// TIA Portal V17 export
// export: Created 2025-03-05T08:02:20.1491544Z, ExportSetting WithDefaults, DisplayName Totally Integrated Automation Portal, DisplayVersion V17 Update 8, DisplayName TIA Portal Openness, DisplayVersion V17 Update 8, DisplayName TIA Portal Version Control Interface, DisplayVersion V17, DisplayName SINAMICS Startdrive Advanced, DisplayVersion V17 SP2, DisplayName SINAMICS Startdrive G110M, G120, G120C, G120D, G120P, G115D, DisplayVersion V17 SP2, DisplayName SINAMICS Startdrive G130, G150, S120, S150, SINAMICS MV, S210, DisplayVersion V17 SP2, DisplayName STEP 7 Professional, DisplayVersion V17 Update 8, DisplayName SINUMERIK ONE STEP 7 Toolbox, DisplayVersion V17 Update 12, DisplayName SINUMERIK 840D sl STEP 7 Toolbox, DisplayVersion V17 Update 12, DisplayName STEP 7 Safety, DisplayVersion V17 Update 6, DisplayName WinCC Advanced, DisplayVersion V17 Update 8
TYPE "GLOBAL_DATA_CLADDING"
// stored: IsFailsafeCompliant false
   STRUCT
      ALL_UNITS_RETURNED : Bool;   // ALL UNITS RETURNED
      ALL_UNITS_OUT_COLL_TRANSF : Bool;   // ALL UNITS OUT COLLISION TRANSFER
      ALL_STATIONS_UNIT_01_RETURNED : Bool;   // ALL UNITS RETURNED / ALL STATIONS UNIT 01 RETURNED
      ALL_STATIONS_UNIT_01_OUT_COLL_TRANSF : Bool;   // ALL UNIT OUT COLLISION TRANSFER / ALL STATIONS UNIT 01 OUT COLLISION TRANSFER
      ALL_STATIONS_UNIT_02_RETURNED : Bool;   // ALL UNITS RETURNED / ALL STATIONS UNIT 02 RETURNED
      ALL_STATIONS_UNIT_02_OUT_COLL_TRANSF : Bool;   // ALL UNIT OUT COLLISION TRANSFER / ALL STATIONS UNIT 02 OUT COLLISION TRANSFER
      ALL_CLAMPED_UNIT_01_ANALOG : Bool;   // ALL CLAMPED / ALL CLAMPED UNIT 01
      ALL_UNCLAMPED_UNIT_01_ANALOG : Bool;   // ALL UNCLAMPED / ALL UNCLAMPED UNIT 01
      ALL_CLAMPED_UNIT_02_ANALOG : Bool;   // ALL CLAMPED / ALL CLAMPED UNIT 02
      ALL_UNCLAMPED_UNIT_02_ANALOG : Bool;   // ALL UNCLAMPED / ALL UNCLAMPED UNIT 02
      CLAMPED_UNCLAMPED_UNIT_01_ANALOG : Bool;   // CLAMPED OR UNCLAMPED / CLAMPED OR UNCLAMPED UNIT 01
      CLAMPED_PARTIAL_CLAMPED_UNIT_01_ANALOG : Bool;   // CLAMPED OR UNCLAMPED / CLAMPED OR PARTIAL CLAMPED UNIT 01
      CLAMPED_UNCLAMPED_UNIT_02_ANALOG : Bool;   // CLAMPED OR UNCLAMPED / CLAMPED OR UNCLAMPED UNIT 02
      CLAMPED_PARTIAL_CLAMPED_UNIT_02_ANALOG : Bool;   // CLAMPED OR UNCLAMPED / CLAMPED OR PARTIAL CLAMPED UNIT 02
      ALL_CLAMPED_UNIT_01 : Bool;   // ALL CLAMPED / ALL CLAMPED UNIT 01
      ALL_UNCLAMPED_UNIT_01 : Bool;   // ALL UNCLAMPED / ALL UNCLAMPED UNIT 01
      ALL_CLAMPED_UNIT_02 : Bool;   // ALL CLAMPED / ALL CLAMPED UNIT 02
      ALL_UNCLAMPED_UNIT_02 : Bool;   // ALL UNCLAMPED / ALL UNCLAMPED UNIT 02
      CLAMPED_UNCLAMPED_UNIT_01 : Bool;   // CLAMPED OR UNCLAMPED / CLAMPED OR UNCLAMPED UNIT 01
      CLAMPED_PARTIAL_CLAMPED_UNIT_01 : Bool;   // CLAMPED OR UNCLAMPED / CLAMPED OR PARTIAL CLAMPED UNIT 01
      CLAMPED_UNCLAMPED_UNIT_02 : Bool;   // CLAMPED OR UNCLAMPED / CLAMPED OR UNCLAMPED UNIT 02
      CLAMPED_PARTIAL_CLAMPED_UNIT_02 : Bool;   // CLAMPED OR UNCLAMPED / CLAMPED OR PARTIAL CLAMPED UNIT 02
      CLAMPED_UNCLAMPED_UNIT_03 : Bool;   // CLAMPED OR UNCLAMPED / CLAMPED OR UNCLAMPED UNIT 03
      CLAMPED_PARTIAL_CLAMPED_UNIT_03 : Bool;   // CLAMPED OR UNCLAMPED / CLAMPED OR PARTIAL CLAMPED UNIT 03
      FIX_IN_UNIT_01_STA_1_UNCLAMPED_ANALOG : Bool;   // FIXTURE IN UNIT 01 LOAD UNLOAD STATION UNCLAMPED ANALOG
      FIX_IN_UNIT_01_STA_1_CLAMPED_ANALOG : Bool;   // FIXTURE IN UNIT 01 LOAD UNLOAD STATION CLAMPED ANALOG
      FIX_IN_UNIT_02_STA_1_UNCLAMPED_ANALOG : Bool;   // FIXTURE IN UNIT 02 LOAD UNLOAD STATION UNCLAMPED ANALOG
      FIX_IN_UNIT_02_STA_1_CLAMPED_ANALOG : Bool;   // FIXTURE IN UNIT 02 LOAD UNLOAD STATION CLAMPED ANALOG
      FIX_IN_UNIT_01_STA_2_UNCLAMPED_ANALOG : Bool;   // FIXTURE IN UNIT 01 SPARE STATION UNCLAMPED ANALOG
      FIX_IN_UNIT_01_STA_2_CLAMPED_ANALOG : Bool;   // FIXTURE IN UNIT 01 SPARE STATION CLAMPED ANALOG
      FIX_IN_UNIT_02_STA_2_UNCLAMPED_ANALOG : Bool;   // FIXTURE IN UNIT 02 SPARE STATION UNCLAMPED ANALOG
      FIX_IN_UNIT_02_STA_2_CLAMPED_ANALOG : Bool;   // FIXTURE UNIT 02 IN SPARE STATION CLAMPED ANALOG
      FIX_IN_UNIT_01_STA_3_UNCLAMPED_ANALOG : Bool;   // FIXTURE IN UNIT 01 CLADDING STATION UNCLAMPED ANALOG
      FIX_IN_UNIT_01_STA_3_CLAMPED_ANALOG : Bool;   // FIXTURE IN UNIT 01 CLADDING STATION CLAMPED ANALOG
      FIX_IN_UNIT_02_STA_3_UNCLAMPED_ANALOG : Bool;   // FIXTURE IN UNIT 02 CLADDING STATION UNCLAMPED ANALOG
      FIX_IN_UNIT_02_STA_3_CLAMPED_ANALOG : Bool;   // FIXTURE IN UNIT 02 CLADDING STATION CLAMPED ANALOG
      FIX_IN_UNIT_01_STA_4_UNCLAMPED_ANALOG : Bool;   // FIXTURE IN UNIT 01 MEASURING/CLEANING STATION UNCLAMPED ANALOG
      FIX_IN_UNIT_01_STA_4_CLAMPED_ANALOG : Bool;   // FIXTURE IN UNIT 01 MEASURING/CLEANING STATION CLAMPED ANALOG
      FIX_IN_UNIT_02_STA_4_UNCLAMPED_ANALOG : Bool;   // FIXTURE IN UNIT 02 MEASURING/CLEANING STATION UNCLAMPED ANALOG
      FIX_IN_UNIT_02_STA_4_CLAMPED_ANALOG : Bool;   // FIXTURE UNIT 02 IN MEASURING/CLEANING STATION CLAMPED ANALOG
      FIX_IN_UNIT_01_STA_1_UNCLAMPED : Bool;   // FIXTURE IN UNIT 01 LOAD UNLOAD STATION UNCLAMPED
      FIX_IN_UNIT_01_STA_1_CLAMPED : Bool;   // FIXTURE IN UNIT 01 LOAD UNLOAD STATION CLAMPED
      FIX_IN_UNIT_02_STA_1_UNCLAMPED : Bool;   // FIXTURE IN UNIT 02 LOAD UNLOAD STATION UNCLAMPED
      FIX_IN_UNIT_02_STA_1_CLAMPED : Bool;   // FIXTURE IN UNIT 02 LOAD UNLOAD STATION CLAMPED
      FIX_IN_UNIT_01_STA_2_UNCLAMPED : Bool;   // FIXTURE IN UNIT 01 SPARE STATION UNCLAMPED
      FIX_IN_UNIT_01_STA_2_CLAMPED : Bool;   // FIXTURE IN UNIT 01 SPARE STATION CLAMPED
      FIX_IN_UNIT_02_STA_2_UNCLAMPED : Bool;   // FIXTURE IN UNIT 02 SPARE STATION UNCLAMPED
      FIX_IN_UNIT_02_STA_2_CLAMPED : Bool;   // FIXTURE UNIT 02 IN SPARE STATION CLAMPED
      FIX_IN_UNIT_01_STA_3_UNCLAMPED : Bool;   // FIXTURE IN UNIT 01 CLADDING STATION UNCLAMPED
      FIX_IN_UNIT_01_STA_3_CLAMPED : Bool;   // FIXTURE IN UNIT 01 CLADDING STATION CLAMPED
      FIX_IN_UNIT_02_STA_3_UNCLAMPED : Bool;   // FIXTURE IN UNIT 02 CLADDING STATION UNCLAMPED
      FIX_IN_UNIT_02_STA_3_CLAMPED : Bool;   // FIXTURE IN UNIT 02 CLADDING STATION CLAMPED
      FIX_IN_UNIT_01_STA_4_UNCLAMPED : Bool;   // FIXTURE IN UNIT 01 MEASURING/CLEANING STATION UNCLAMPED
      FIX_IN_UNIT_01_STA_4_CLAMPED : Bool;   // FIXTURE IN UNIT 01 MEASURING/CLEANING STATION CLAMPED
      FIX_IN_UNIT_02_STA_4_UNCLAMPED : Bool;   // FIXTURE IN UNIT 02 MEASURING/CLEANING STATION UNCLAMPED
      FIX_IN_UNIT_02_STA_4_CLAMPED : Bool;   // FIXTURE UNIT 02 IN MEASURING/CLEANING STATION CLAMPED
      FIX_IN_UNIT_03_STA_MEAS_UNCLAMPED : Bool;   // FIXTURE IN UNIT 03 MEASURING STATION UNCLAMPED ANALOG
      FIX_IN_UNIT_03_STA_MEAS_CLAMPED : Bool;   // FIXTURE UNIT 03 IN MEASURING STATION CLAMPED ANALOG
      FIX_IN_UNIT_01_STA_0_ANY_CALIBRATION_MISS : Bool;   // FIXTURE IN UNIT 01 STATION 0 ANY CALIBRATION MISSING
      FIX_IN_UNIT_02_STA_0_ANY_CALIBRATION_MISS : Bool;   // FIXTURE IN UNIT 02 STATION 0 ANY CALIBRATION MISSING
      UNIT_01_ANY_FIX_CALIBRATION_MISS : Bool;   // UNIT 01 ANY FIXTURE CALIBRATION MISSING
      UNIT_02_ANY_FIX_CALIBRATION_MISS : Bool;   // UNIT 02 ANY FIXTURE CALIBRATION MISSING
      MACHINE_ANY_FIX_CALIBRATION_MISS : Bool;   // MACHINE ANY FIXTURE CALIBRATION MISSING
      ALL_FULL_DEPTH : Bool;   // ALL FULL DEPTH
      ALL_FULL_DEPTH_PULSE : Bool;   // ALL FULL DEPTH PULSE
      ALL_FULL_DEPTH_UNIT_01 : Bool;   // ALL FULL DEPTH / ALL FULL DEPTH UNIT 01
      ALL_FULL_DEPTH_PULSE_UNIT_01 : Bool;   // ALL FULL DEPTH PULSE / ALL FULL DEPTH PULSE UNIT 01
      ALL_FULL_DEPTH_UNIT_02 : Bool;   // ALL FULL DEPTH / ALL FULL DEPTH UNIT 02
      ALL_FULL_DEPTH_PULSE_UNIT_02 : Bool;   // ALL FULL DEPTH PULSE / ALL FULL DEPTH PULSE UNIT 02
      ALL_FULL_DEPTH_UNIT_03 : Bool;   // ALL FULL DEPTH / ALL FULL DEPTH UNIT 03
      ALL_FULL_DEPTH_PULSE_UNIT_03 : Bool;   // ALL FULL DEPTH PULSE / ALL FULL DEPTH PULSE UNIT 03
      RESET_FULL_DEPTH_UNIT_01_FIXT_1 : Bool;   // RESET FULL DEPTH / RESET FULL DEPTH UNIT 01 FIXTURE 1
      RESET_FULL_DEPTH_PULSE_UNIT_01_FIXT_1 : Bool;   // RESET FULL DEPTH PULSE / RESET FULL DEPTH PULSE UNIT 01 FIXTURE 1
      RESET_FULL_DEPTH_UNIT_01_FIXT_2 : Bool;   // RESET FULL DEPTH UNIT 01 FIXTURE 2
      RESET_FULL_DEPTH_PULSE_UNIT_01_FIXT_2 : Bool;   // RESET FULL DEPTH PULSE UNIT 01 FIXTURE 2
      RESET_FULL_DEPTH_UNIT_01_FIXT_3 : Bool;   // RESET FULL DEPTH / RESET FULL DEPTH UNIT 01 FIXTURE 3
      RESET_FULL_DEPTH_PULSE_UNIT_01_FIXT_3 : Bool;   // RESET FULL DEPTH PULSE / RESET FULL DEPTH PULSE UNIT 01 FIXTURE 3
      RESET_FULL_DEPTH_UNIT_01_FIXT_4 : Bool;   // RESET FULL DEPTH UNIT 01 FIXTURE 4
      RESET_FULL_DEPTH_PULSE_UNIT_01_FIXT_4 : Bool;   // RESET FULL DEPTH PULSE UNIT 01 FIXTURE 4
      RESET_FULL_DEPTH_UNIT_02_FIXT_1 : Bool;   // RESET FULL DEPTH / RESET FULL DEPTH UNIT 02 FIXTURE 1
      RESET_FULL_DEPTH_PULSE_UNIT_02_FIXT_1 : Bool;   // RESET FULL DEPTH PULSE / RESET FULL DEPTH PULSE UNIT 02 FIXTURE 1
      RESET_FULL_DEPTH_UNIT_02_FIXT_2 : Bool;   // RESET FULL DEPTH / RESET FULL DEPTH UNIT 02 FIXTURE 2
      RESET_FULL_DEPTH_PULSE_UNIT_02_FIXT_2 : Bool;   // RESET FULL DEPTH PULSE / RESET FULL DEPTH PULSE UNIT 02 FIXTURE 2
      RESET_FULL_DEPTH_UNIT_02_FIXT_3 : Bool;   // RESET FULL DEPTH / RESET FULL DEPTH UNIT 02 FIXTURE 3
      RESET_FULL_DEPTH_PULSE_UNIT_02_FIXT_3 : Bool;   // RESET FULL DEPTH PULSE / RESET FULL DEPTH PULSE UNIT 02 FIXTURE 3
      RESET_FULL_DEPTH_UNIT_02_FIXT_4 : Bool;   // RESET FULL DEPTH / RESET FULL DEPTH UNIT 02 FIXTURE 4
      RESET_FULL_DEPTH_PULSE_UNIT_02_FIXT_4 : Bool;   // RESET FULL DEPTH PULSE / RESET FULL DEPTH PULSE UNIT 02 FIXTURE 4
      RESET_FULL_DEPTH_UNIT_03_FIXT_1 : Bool;   // RESET FULL DEPTH / RESET FULL DEPTH UNIT 01 FIXTURE 1
      RESET_FULL_DEPTH_PULSE_UNIT_03_FIXT_1 : Bool;   // RESET FULL DEPTH PULSE / RESET FULL DEPTH PULSE UNIT 01 FIXTURE 1
      NO_MACHINE_CYCLE_RUN_P : Bool;   // NO CYCLE MACHINE RUN PROGRAM / NO MACHINE CYCLE RUNNING PULSE
      ANY_MACHINE_CYCLE_RUN_P : Bool;   // ANY MACHINE CYCLE RUN PROGRAM / ANY MACHINE CYCLE RUNNING PULSE
      NO_MACHINE_CYCLE_RUN_UNIT_01_P : Bool;   // NO CYCLE MACHINE RUN PROGRAM / NO MACHINE CYCLE RUNNING UNIT 01 PULSE
      ANY_UNIT_01_CYCLE_RUN_P : Bool;   // ANY MACHINE CYCLE RUN PROGRAM / ANY UNIT 01 CYCLE RUNNING PULSE
      NO_MACHINE_CYCLE_RUN_UNIT_02_P : Bool;   // NO CYCLE MACHINE RUN PROGRAM / NO MACHINE CYCLE RUNNING UNIT 02 PULSE
      ANY_UNIT_02_CYCLE_RUN_P : Bool;   // ANY MACHINE CYCLE RUN PROGRAM / ANY UNIT 02 CYCLE RUNNING PULSE
      NO_MACHINE_CYCLE_RUN_UNIT_03_P : Bool;   // NO CYCLE MACHINE RUN PROGRAM / NO MACHINE CYCLE RUNNING UNIT 03 PULSE
      ANY_UNIT_03_CYCLE_RUN_P : Bool;   // ANY MACHINE CYCLE RUN PROGRAM / ANY UNIT 03 CYCLE RUNNING PULSE
      NO_MACHINE_CYCLE_RUN_HOPPER_UNIT_01_P : Bool;   // NO CYCLE MACHINE RUN PROGRAM / NO MACHINE CYCLE RUNNING HOPPER UNIT 01 PULSE
      ANY_HOPPER_UNIT_01_CYCLE_RUN_P : Bool;   // ANY MACHINE CYCLE RUN PROGRAM / ANY HOPPER UNIT 01 CYCLE RUNNING PULSE
      NO_MACHINE_CYCLE_RUN_HOPPER_UNIT_02_P : Bool;   // NO CYCLE MACHINE RUN PROGRAM / NO MACHINE CYCLE RUNNING HOPPER UNIT 02 PULSE
      ANY_HOPPER_UNIT_02_CYCLE_RUN_P : Bool;   // ANY MACHINE CYCLE RUN PROGRAM / ANY HOPPER UNIT 02 CYCLE RUNNING PULSE
      FIX_IN_U_01_STA_1_ANY_FIX_SEQ_RUN : Bool;   // (GLOBAL BITS) COOLANT ON UNIT 01R / FIXTURE IN UNIT 01 STATION 1 RUNING ANY SEQUENCE
      FIX_IN_U_01_STA_2_ANY_FIX_SEQ_RUN : Bool;   // (GLOBAL BITS) COOLANT UNIT 01R WAIT FOR FILL TOOL / FIXTURE IN UNIT 01 STATION 2 RUNING ANY SEQUENCE
      FIX_IN_U_01_STA_3_ANY_FIX_SEQ_RUN : Bool;   // (GLOBAL BITS) COOLANT ON UNIT 01L / FIXTURE IN UNIT 01 STATION 3 RUNING ANY SEQUENCE
      FIX_IN_U_01_STA_4_ANY_FIX_SEQ_RUN : Bool;   // (GLOBAL BITS) COOLANT UNIT 01L WAIT FOR FILL TOOL / FIXTURE IN UNIT 01 STATION 4 RUNING ANY SEQUENCE
      FIX_IN_U_02_STA_1_ANY_FIX_SEQ_RUN : Bool;   // (GLOBAL BITS) COOLANT SP11 ON / FIXTURE IN UNIT 02 STATION 1 RUNING ANY SEQUENCE
      FIX_IN_U_02_STA_2_ANY_FIX_SEQ_RUN : Bool;   // (GLOBAL BITS) COOLANT SP12 ON / FIXTURE IN UNIT 02 STATION 2 RUNING ANY SEQUENCE
      FIX_IN_U_02_STA_3_ANY_FIX_SEQ_RUN : Bool;   // (GLOBAL BITS) COOLANT SP13 ON / FIXTURE IN UNIT 02 STATION 3 RUNING ANY SEQUENCE
      FIX_IN_U_02_STA_4_ANY_FIX_SEQ_RUN : Bool;   // (GLOBAL BITS) COOLANT SP14 ON / FIXTURE IN UNIT 02 STATION 4 RUNING ANY SEQUENCE
      FIX_IN_U_01_STA_1_PART_PRESENT : Bool;   // (GLOBAL BITS) COOLANT SP21 ON / FIXTURE IN UNIT 01 STATION 1 PART PRESENT
      FIX_IN_U_01_STA_2_PART_PRESENT : Bool;   // (GLOBAL BITS) COOLANT SP21 ON / FIXTURE IN UNIT 01 STATION 2 PART PRESENT
      FIX_IN_U_01_STA_3_PART_PRESENT : Bool;   // (GLOBAL BITS) COOLANT SP21 ON / FIXTURE IN UNIT 01 STATION 3 PART PRESENT
      FIX_IN_U_01_STA_4_PART_PRESENT : Bool;   // (GLOBAL BITS) COOLANT SP21 ON / FIXTURE IN UNIT 01 STATION 4 PART PRESENT
      FIX_IN_U_02_STA_1_PART_PRESENT : Bool;   // (GLOBAL BITS) COOLANT SP21 ON / FIXTURE IN UNIT 02 STATION 1 PART PRESENT
      FIX_IN_U_02_STA_2_PART_PRESENT : Bool;   // (GLOBAL BITS) COOLANT SP21 ON / FIXTURE IN UNIT 02 STATION 2 PART PRESENT
      FIX_IN_U_02_STA_3_PART_PRESENT : Bool;   // (GLOBAL BITS) COOLANT SP21 ON / FIXTURE IN UNIT 02 STATION 3 PART PRESENT
      FIX_IN_U_02_STA_4_PART_PRESENT : Bool;   // (GLOBAL BITS) COOLANT SP21 ON / FIXTURE IN UNIT 02 STATION 4 PART PRESENT
      U01_RN_CYCLE_PART_TYPE : Bool;   // UNIT 01 R-N CYCLE PART TYPE
      U01_NR_CYCLE_PART_TYPE : Bool;   // UNIT 01 N-R CYCLE PART TYPE
      U02_RN_CYCLE_PART_TYPE : Bool;   // UNIT 02 R-N CYCLE PART TYPE
      U02_NR_CYCLE_PART_TYPE : Bool;   // UNIT 02 N-R CYCLE PART TYPE
      ANY_MACHINE_CYCLE_RUN : Bool;   // ANY MACHINE CYCLE RUN / ANY MACHINE CYCLE RUNNING
      ANY_UNIT_01_CYCLE_RUN : Bool;   // ANY MACHINE CYCLE RUN / ANY UNIT 01 CYCLE RUNNING
      ANY_UNIT_02_CYCLE_RUN : Bool;   // ANY MACHINE CYCLE RUN / ANY UNIT 02 CYCLE RUNNING
      ANY_UNIT_03_CYCLE_RUN : Bool;   // ANY MACHINE CYCLE RUN / ANY UNIT 03 CYCLE RUNNING
      ANY_HOPPER_UNIT_01_CYCLE_RUN : Bool;   // ANY MACHINE CYCLE RUN / ANY HOPPER UNIT 01 CYCLE RUNNING
      ANY_HOPPER_UNIT_02_CYCLE_RUN : Bool;   // ANY MACHINE CYCLE RUN / ANY HOPPER UNIT 02 CYCLE RUNNING
      UNIT_01_ST_0_ANY_CYCLE_ACTIVE : Bool;   // STATION 1 ANY CYCLE ACTIVE / UNIT 01 STATION 0 ANY CYCLE ACTIVE
      UNIT_01_ST_1_ANY_CYCLE_ACTIVE : Bool;   // STATION 2 ANY CYCLE ACTIVE / UNIT 01 STATION 1 ANY CYCLE ACTIVE
      UNIT_01_ST_2_ANY_CYCLE_ACTIVE : Bool;   // STATION 3 ANY CYCLE ACTIVE / UNIT 01 STATION 2 ANY CYCLE ACTIVE
      UNIT_01_ST_3_ANY_CYCLE_ACTIVE : Bool;   // STATION 4 ANY CYCLE ACTIVE / UNIT 01 STATION 3 ANY CYCLE ACTIVE
      UNIT_01_ST_4_ANY_CYCLE_ACTIVE : Bool;   // STATION 5 ANY CYCLE ACTIVE / UNIT 01 STATION 4 ANY CYCLE ACTIVE
      UNIT_02_ST_0_ANY_CYCLE_ACTIVE : Bool;   // STATION 6 ANY CYCLE ACTIVE / UNIT 02 STATION 0 ANY CYCLE ACTIVE
      UNIT_02_ST_1_ANY_CYCLE_ACTIVE : Bool;   // STATION 7 ANY CYCLE ACTIVE / UNIT 02 STATION 1 ANY CYCLE ACTIVE
      UNIT_02_ST_2_ANY_CYCLE_ACTIVE : Bool;   // STATION 8 ANY CYCLE ACTIVE / UNIT 02 STATION 2 ANY CYCLE ACTIVE
      UNIT_02_ST_3_ANY_CYCLE_ACTIVE : Bool;   // STATION 9 ANY CYCLE ACTIVE / UNIT 02 STATION 3 ANY CYCLE ACTIVE
      UNIT_02_ST_4_ANY_CYCLE_ACTIVE : Bool;   // STATION 10 ANY CYCLE ACTIVE / UNIT 02 STATION 4 ANY CYCLE ACTIVE
      UNIT_03_ANY_CYCLE_ACTIVE : Bool;   // STATION 11 ANY CYCLE ACTIVE / UNIT 03 ANY CYCLE ACTIVE
      UNIT_12_ANY_CYCLE_ACTIVE : Bool;   // STATION 12 ANY CYCLE ACTIVE / UNIT 12 ANY CYCLE ACTIVE
      ANY_CHANNEL_MG1_RUN : Bool;   // TRANSFER ANY CYCLE ACTIVE / ANY CHANNEL MODE GROUP 1 RUNNING
      ANY_CHANNEL_MG2_RUN : Bool;   // ANY CHANNEL MODE GROUP 2 RUNNING
      ANY_PART_CYCLE_RUN : Bool;   // ANY MACHINE PART CYCLE RUN / ANY MACHINE PART CYCLE RUNNING
      UNIT_01_ST_0_PART_CYCLE_ACTIVE : Bool;   // STATION 1 PART CYCLE ACTIVE / UNIT 01 STATION 0 PART CYCLE ACTIVE
      UNIT_01_ST_1_PART_CYCLE_ACTIVE : Bool;   // STATION 2 PART CYCLE ACTIVE / UNIT 01 STATION 1 PART CYCLE ACTIVE
      UNIT_01_ST_2_PART_CYCLE_ACTIVE : Bool;   // STATION 3 PART CYCLE ACTIVE / UNIT 01 STATION 2 PART CYCLE ACTIVE
      UNIT_01_ST_3_PART_CYCLE_ACTIVE : Bool;   // STATION 4 PART CYCLE ACTIVE / UNIT 01 STATION 3 PART CYCLE ACTIVE
      UNIT_01_ST_4_PART_CYCLE_ACTIVE : Bool;   // STATION 5 PART CYCLE ACTIVE / UNIT 01 STATION 4 PART CYCLE ACTIVE
      UNIT_02_ST_0_PART_CYCLE_ACTIVE : Bool;   // STATION 6 PART CYCLE ACTIVE / UNIT 02 STATION 0 PART CYCLE ACTIVE
      UNIT_02_ST_1_PART_CYCLE_ACTIVE : Bool;   // STATION 7 PART CYCLE ACTIVE / UNIT 02 STATION 1 PART CYCLE ACTIVE
      UNIT_02_ST_2_PART_CYCLE_ACTIVE : Bool;   // STATION 8 PART CYCLE ACTIVE / UNIT 02 STATION 2 PART CYCLE ACTIVE
      UNIT_02_ST_3_PART_CYCLE_ACTIVE : Bool;   // STATION 9 PART CYCLE ACTIVE / UNIT 02 STATION 3 PART CYCLE ACTIVE
      UNIT_02_ST_4_PART_CYCLE_ACTIVE : Bool;   // STATION 10 PART CYCLE ACTIVE / UNIT 02 STATION 4 PART CYCLE ACTIVE
      UNIT_03_PART_CYCLE_ACTIVE : Bool;   // STATION 11 PART CYCLE ACTIVE / UNIT 03 PART CYCLE ACTIVE
      UNIT_12_PART_CYCLE_ACTIVE : Bool;   // STATION 12 PART CYCLE ACTIVE / UNIT 12 PART CYCLE ACTIVE
      MACHINE_AT_HOME_POSITION : Bool;   // MACHINE AT HOME POSITION
      UNIT_01_AT_HOME_POS : Bool;   // STATION 1 AT HOME POSITION / UNIT 01 AT HOME POSITION
      UNIT_02_AT_HOME_POS : Bool;   // STATION 2 AT HOME POSITION / UNIT 02 AT HOME POSITION
      UNIT_03_AT_HOME_POS : Bool;   // STATION 3 AT HOME POSITION / UNIT 03 AT HOME POSITION
      UNIT_01_STA_0_AT_PARTIAL_HOME_POS : Bool;   // STATION 4 AT HOME POSITION / UNIT 01 STATION 0 AT PARTIAL HOME POSITION
      UNIT_01_STA_0_AT_HOME_POS : Bool;   // STATION 4 AT HOME POSITION / UNIT 01 STATION 0 AT HOME POSITION
      UNIT_01_STA_1_AT_HOME_POS : Bool;   // STATION 5 AT HOME POSITION / UNIT 01 STATION 1 AT HOME POSITION
      UNIT_01_STA_2_AT_HOME_POS : Bool;   // STATION 6 AT HOME POSITION / UNIT 01 STATION 2 AT HOME POSITION
      UNIT_01_STA_3_AT_HOME_POS : Bool;   // STATION 7 AT HOME POSITION / UNIT 01 STATION 3 AT HOME POSITION
      UNIT_01_STA_4_AT_HOME_POS : Bool;   // STATION 8 AT HOME POSITION / UNIT 01 STATION 4 AT HOME POSITION
      UNIT_02_STA_0_AT_PARTIAL_HOME_POS : Bool;   // STATION 4 AT HOME POSITION / UNIT 01 STATION 0 AT PARTIAL HOME POSITION
      UNIT_02_STA_0_AT_HOME_POS : Bool;   // STATION 9 AT HOME POSITION / UNIT 02 STATION 0 AT HOME POSITION
      UNIT_02_STA_1_AT_HOME_POS { ExternalWritable := 'False'} : Bool;   // STATION 10 AT HOME POSITION / UNIT 02 STATION 1 AT HOME POSITION
      UNIT_02_STA_2_AT_HOME_POS : Bool;   // STATION 11 AT HOME POSITION / UNIT 02 STATION 2 AT HOME POSITION
      UNIT_02_STA_3_AT_HOME_POS : Bool;   // STATION 12 AT HOME POSITION / UNIT 02 STATION 3 AT HOME POSITION
      UNIT_02_STA_4_AT_HOME_POS : Bool;   // STATION 13 AT HOME POSITION / UNIT 02 STATION 4 AT HOME POSITION
      UNIT_SPARE_AT_HOME_POS : Bool;   // STATION 14 AT HOME POSITION / UNIT SPARE AT HOME POSITION
      UNIT_01_ANY_M_OPEN_DOOR_REQ : Bool;   // UNIT 01 ANY M TO OPEN ANY DOOR ACTIVE
      UNIT_02_ANY_M_OPEN_DOOR_REQ : Bool;   // UNIT 02 ANY M TO OPEN ANY DOOR ACTIVE
      AUX0 : Bool;   // AUXILIARY 0
      AUX1 : Bool;   // AUXILIARY 1
      AUX2 : Bool;   // AUXILIARY 2
      AUX3 : Bool;   // AUXILIARY 3
      AUX4 : Bool;   // AUXILIARY 4
      AUX5 : Bool;   // AUXILIARY 5
      AUX6 : Bool;   // AUXILIARY 6
      AUX7 : Bool;   // AUXILIARY 7
      AUX8 : Bool;   // AUXILIARY 8
      AUX9 : Bool;   // AUXILIARY 9
      AUX10 : Bool;   // AUXILIARY 10
      AUX11 : Bool;   // AUXILIARY 11
      AUX12 : Bool;   // AUXILIARY 12
      AUX13 : Bool;   // AUXILIARY 13
      AUX14 : Bool;   // AUXILIARY 14
      AUX15 : Bool;   // AUXILIARY 15
      AUX16 : Bool;   // AUXILIARY 16
      AUX17 : Bool;   // AUXILIARY 17
      AUX18 : Bool;   // AUXILIARY 18
      AUX19 : Bool;   // AUXILIARY 19
      AUX20 : Bool;   // AUXILIARY 20
   END_STRUCT;
END_TYPE
